FUNCTION_BLOCK AUS_D_FF (* Data latch (d) flip flop *)
  (* Standard: 61499-1 Annex A; Description: Copyright (c) 2017 fortiss GmbH, HR Agrartechnik GmbH This program and the accompanying materials are made available under the terms of the Eclipse Public License 2.0 which is available at https://www.eclipse.org/legal/epl-2.0/ SPDX-License-Identifier: EPL-2.0 *)
  (* Version 1.0, 2026-05-15, Franz Höpfinger, HR Agrartechnik GmbH, Initial Version *)
  PACKAGE adapter::events::unidirectional;
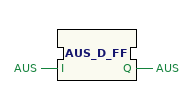
  SOCKETS
    I : adapter::types::unidirectional::AUS; (* Value to latch *)
  END_SOCKETS
  PLUGS
    Q : adapter::types::unidirectional::AUS; (* Latched value *)
  END_PLUGS
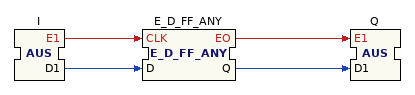
  FBS
    E_D_FF_ANY : iec61499::events::E_D_FF_ANY;
  END_FBS
  EVENT_CONNECTIONS
    I.E1 TO E_D_FF_ANY.CLK;
    E_D_FF_ANY.EO TO Q.E1;
  END_CONNECTIONS
  DATA_CONNECTIONS
    I.D1 TO E_D_FF_ANY.D;
    E_D_FF_ANY.Q TO Q.D1;
  END_CONNECTIONS
END_FUNCTION_BLOCK
